FUNCTION_BLOCK FB_LightControl implements I_LightControl
VAR_INPUT
END_VAR
VAR_OUTPUT
END_VAR
VAR
END_VAR

{warning 'add method implementation'}
METHOD M_Reset : BOOL
END_METHOD

{warning 'add method implementation'}
METHOD M_Set : BOOL
END_METHOD

{warning 'add property implementation'}
PROPERTY nAddress : DINT
GET
END_GET
SET
END_SET
END_PROPERTY

{warning 'add property implementation'}
PROPERTY nIlluminance : REAL
GET
END_GET
SET
END_SET
END_PROPERTY

END_FUNCTION_BLOCK

(* stored: Version 1.1.0.1, ProductVersion 3.1.4022.18
   POU FB_LightControl: Id {076fe08a-3174-4c6e-92fc-678cc5e96626}, SpecialFunc None
   Method M_Reset: Id {734b9f71-48e0-4337-9e75-de2d5e42786a}
   Method M_Set: Id {f50a4cd7-4d1a-40a6-97ee-2fa23772c497}
   Property nAddress: Id {980c8121-a09f-4a3d-b6fa-7c634df64e4e}
   Get Get: Id {8d694bfc-73ac-4af4-b25d-03a0bce9cb5e}
   Set Set: Id {f6b678ee-7526-4c84-a48f-772d4c96c787}
   Property nIlluminance: Id {fdd7aad5-6cd9-4f6a-80dc-2bfcd6574726}
   Get Get: Id {00b38a78-40ea-4ca0-81f5-9ee364f795a7}
   Set Set: Id {2ed18869-62a1-46be-99bc-1a6bcbfd90ea} *)
